// TIA Portal V19 export
ORGANIZATION_BLOCK "Main"   // OB1, LAD, ProgramCycle
TITLE = "Main Program Sweep (Cycle)"
{ S7_Optimized_Access := 'TRUE' }
// stored: SetENOAutomatically false
   VAR_INPUT
      Initial_Call : Bool;   // Initial call of this OB
      Remanence : Bool;   // =True, if remanent data are available
   END_VAR
   VAR_TEMP   // added for the SCL form of the ladder/FBD networks
      _w1 : Bool;
   END_VAR
BEGIN

REGION Network 1: Homing Vertical
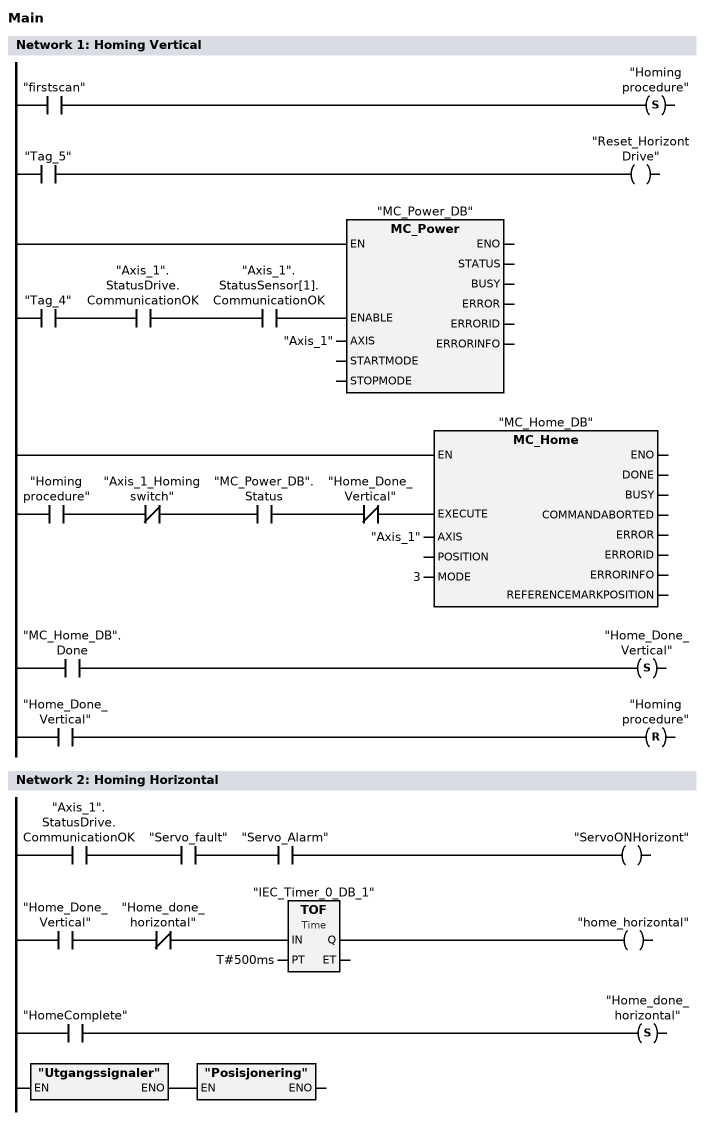
   RUNG wire#powerrail
      Contact( "firstscan" )
      S_Coil( "Homing procedure" )
   END_RUNG
   RUNG wire#powerrail
      Contact( "Tag_5" )
      Coil( "Reset_HorizontDrive" )
   END_RUNG
   RUNG wire#powerrail
      "MC_Power_DB".MC_Power(Enable := wire#w1, Axis := "Axis_1", StartMode :=, StopMode :=, Status =>, Busy =>, Error =>, ErrorID =>, ErrorInfo =>)
   END_RUNG
   RUNG wire#powerrail
      Contact( "Tag_4" )
      Contact( "Axis_1".StatusDrive.CommunicationOK )
      Contact( "Axis_1".StatusSensor[1].CommunicationOK )
   END_RUNG wire#w1
   RUNG wire#powerrail
      "MC_Home_DB".MC_Home(Execute := wire#w2, Axis := "Axis_1", Position :=, Mode := 3, Done =>, Busy =>, CommandAborted =>, Error =>, ErrorID =>, ErrorInfo =>, ReferenceMarkPosition =>)
   END_RUNG
   RUNG wire#powerrail
      Contact( "Homing procedure" )
      I_Contact( "Axis_1_Homing switch" )
      Contact( "MC_Power_DB".Status )
      I_Contact( "Home_Done_Vertical" )
   END_RUNG wire#w2
   RUNG wire#powerrail
      Contact( "MC_Home_DB".Done )
      S_Coil( "Home_Done_Vertical" )
   END_RUNG
   RUNG wire#powerrail
      Contact( "Home_Done_Vertical" )
      R_Coil( "Homing procedure" )
   END_RUNG
   // the same network as SCL:
   IF "firstscan" THEN "Homing procedure" := TRUE; END_IF;
   "Reset_HorizontDrive" := "Tag_5";
   "MC_Power_DB"(Enable := "Tag_4" AND "Axis_1".StatusDrive.CommunicationOK AND "Axis_1".StatusSensor[1].CommunicationOK,   // MC_Power
                 Axis := "Axis_1");
   "MC_Home_DB"(Execute := "Homing procedure" AND NOT "Axis_1_Homing switch" AND "MC_Power_DB".Status AND NOT "Home_Done_Vertical",   // MC_Home
                Axis := "Axis_1",
                Mode := 3);
   IF "MC_Home_DB".Done THEN "Home_Done_Vertical" := TRUE; END_IF;
   IF "Home_Done_Vertical" THEN "Homing procedure" := FALSE; END_IF;
END_REGION

REGION Network 2: Homing Horizontal
   RUNG wire#powerrail
      Contact( "Axis_1".StatusDrive.CommunicationOK )
      Contact( "Servo_fault" )
      Contact( "Servo_Alarm" )
      Coil( "ServoONHorizont" )
   END_RUNG
   RUNG wire#powerrail
      Contact( "Home_Done_Vertical" )
      I_Contact( "Home_done_horizontal" )
      { S7_Templates := "time_type := Time" } "IEC_Timer_0_DB_1".TOF(pt := T#500ms, et =>)
      Coil( "home_horizontal" )
   END_RUNG
   RUNG wire#powerrail
      Contact( "HomeComplete" )
      S_Coil( "Home_done_horizontal" )
   END_RUNG
   RUNG wire#powerrail
      "Utgangssignaler"()
      "Posisjonering"()
   END_RUNG
   // the same network as SCL:
   "ServoONHorizont" := "Axis_1".StatusDrive.CommunicationOK AND "Servo_fault" AND "Servo_Alarm";
   "IEC_Timer_0_DB_1".TOF(IN := "Home_Done_Vertical" AND NOT "Home_done_horizontal", PT := T#500ms);
   "home_horizontal" := "IEC_Timer_0_DB_1".Q;
   IF "HomeComplete" THEN "Home_done_horizontal" := TRUE; END_IF;
   "Utgangssignaler"(ENO => #_w1);
   IF #_w1 THEN "Posisjonering"(); END_IF;
END_REGION
END_ORGANIZATION_BLOCK
